TYPE ST_TempLoad :
STRUCT
	stTempCmd: ST_TempLoad_Cmd;
	stTempState: ST_TempLoad_State;
END_STRUCT
END_TYPE

(* stored: Version 1.1.0.1, ProductVersion 3.1.0.26
   DUT ST_TempLoad: Id {0e0b134f-eb0f-42cc-b524-4d4227e3d9cb} *)
